FUNCTION_BLOCK FB_StringBuilder
VAR
	sContent : STRING; // Store temporary strings;
END_VAR

METHOD Append : REFERENCE TO FB_StringBuilder
VAR_INPUT
	sText : STRING;
END_VAR
sContent := CONCAT(STR1 := sContent, STR2 := sText);
Append REF= THIS^;
END_METHOD

METHOD Clear : REFERENCE TO FB_StringBuilder
VAR_INPUT
END_VAR
sContent := '';
Clear REF= THIS^;
END_METHOD

METHOD ToString : STRING
VAR_INPUT
END_VAR
ToString := sContent; // return internal content
END_METHOD

END_FUNCTION_BLOCK

(* stored: Version 1.1.0.1, ProductVersion 3.1.4024.12
   POU FB_StringBuilder: Id {2318978f-2a07-4c2a-9672-0a22ff2518ba}, SpecialFunc None
   Method Append: Id {6e8f5106-1c12-4e90-b69c-c5893b2f0211}
   Method Clear: Id {c40fe4e4-01da-40b5-9278-42da0354d992}
   Method ToString: Id {f593a77f-74af-4630-a72a-39ec9153b6cc} *)
